{attribute 'enable_dynamic_creation'}
{attribute 'no_explicit_call' := 'do not call this FB directly'}
FUNCTION_BLOCK PUBLIC ABSTRACT FileSystemEntry IMPLEMENTS I_FileSystemEntry, I_Disposable
VAR
	_path : FilePath;	
END_VAR

METHOD Dispose
__DELETE(THIS);
END_METHOD

METHOD FB_init : BOOL
VAR_INPUT
	bInitRetains : BOOL; // if TRUE, the retain variables are initialized (warm start / cold start)
	bInCopyCode : BOOL;  // if TRUE, the instance afterwards gets moved into the copy code (online change)
	Path : FilePath;
END_VAR
THIS^._path := PathCorrection(Path);
END_METHOD

PROPERTY PUBLIC IsDirectory : BOOL
GET
IsDirectory := FALSE;
END_GET
END_PROPERTY

PROPERTY PUBLIC IsFile : BOOL
GET
IsFile := FALSE;
END_GET
END_PROPERTY

PROPERTY PUBLIC IsNull : BOOL
GET
IsNull := FALSE;
END_GET
END_PROPERTY

PROPERTY Path : FilePath
GET
Path := _path;
END_GET
END_PROPERTY

METHOD PRIVATE PathCorrection : FilePath
VAR_INPUT
	PathToCheck : FilePath;
END_VAR
IF (PathToCheck = '') THEN
	PathCorrection := '.\';
	RETURN;
END_IF

IF (RIGHT(PathToCheck, 1) <> '\') THEN
	PathCorrection := CONCAT(PathToCheck, '\');
	RETURN;
END_IF

PathCorrection := PathToCheck;
END_METHOD

END_FUNCTION_BLOCK

(* stored: Version 1.1.0.1, ProductVersion 3.1.4024.9
   POU FileSystemEntry: Id {88d5ad2d-c055-4393-82a7-d01f5d3379eb}, SpecialFunc None
   Folder Constructor: Id {700ef6a9-b5fe-4af4-b7d6-effcf0a5f087}
   Folder Private: Id {27846fc7-15f2-4e94-a698-4cb4e694175c}
   Method Dispose: Id {a35e5125-c9c9-47fb-b996-f8c06aa27213}
   Method FB_init: Id {ba74ccb0-59d7-475b-b89b-2bd4ca370d16}
   Property IsDirectory: Id {9103648a-0894-4df3-96d0-863e5ce067d1}
   Get Get: Id {fd87137c-f12a-4725-a347-fe3049c677a1}
   Property IsFile: Id {6320f1ff-661e-46b3-b17c-fb38add9c551}
   Get Get: Id {f18eea18-e04f-41a1-a648-f4fc3a36c1a1}
   Property IsNull: Id {47d25653-6e57-40d0-b86d-f3316f0cf71d}
   Get Get: Id {108520d4-36ce-4c13-bc0f-19dd17918fc0}
   Property Path: Id {0c75e418-fa36-4cba-8aca-9011fc540de4}
   Get Get: Id {3122b97c-7417-4d2b-a123-627a45757fa4}
   Method PathCorrection: Id {07ef579f-3cb5-4875-a980-765197adebd7} *)
